// TIA Portal V17 export
// export: Created 2024-09-02T12:50:23.8118301Z, ExportSetting WithDefaults, DisplayName Totally Integrated Automation Portal, DisplayVersion V17, DisplayName TIA Portal Openness, DisplayVersion V17, DisplayName TIA Portal Version Control Interface, DisplayVersion V17, DisplayName STEP 7 Professional, DisplayVersion V17, DisplayName STEP 7 Safety, DisplayVersion V17, DisplayName WinCC Professional, DisplayVersion V17
DATA_BLOCK "DBi_Aveva_OP70_1"   // DB701
{ S7_Optimized_Access := 'FALSE' }
VERSION : 0.1
// stored: AutoNumber false, DBAccessibleFromOPCUA true, IsOnlyStoredInLoadMemory false, IsWriteProtectedInAS false
   VAR
      SettingSpecyfications : Struct
         Global { S7_SetPoint := 'True'} : "Aveva_Data_Spec";   // General data for all Stations
         Station : Struct   // Specific data (depending on the tools installed on the station)
            Empty : "Aveva_Empty_Spec";
         END_STRUCT;
      END_STRUCT;
      Result : Struct
         Global : "Aveva_Data_Result";   // General data for all Stations
         Station : Struct   // Specific data (depending on the tools installed on the station)
            Empty : "Aveva_Empty_Result";
         END_STRUCT;
      END_STRUCT;
      init : Struct
         SettingSpecyfications : Struct
            Global { S7_SetPoint := 'True'} : "Aveva_Data_Spec";   // General data for all Stations
            Station : Struct   // Specific data (depending on the tools installed on the station)
               Empty : "Aveva_Empty_Spec";
            END_STRUCT;
         END_STRUCT;
         Result : Struct
            Global : "Aveva_Data_Result";   // General data for all Stations
            Station : Struct   // Specific data (depending on the tools installed on the station)
               Empty : "Aveva_Empty_Result";
            END_STRUCT;
         END_STRUCT;
      END_STRUCT;
   END_VAR
BEGIN
END_DATA_BLOCK
